// TIA Portal V17 export
// export: Created 2022-04-06T07:28:41.6787381Z, ExportSetting WithDefaults, DisplayName Totally Integrated Automation Portal, DisplayVersion V17, DisplayName TIA Portal Openness, DisplayVersion V17, DisplayName TIA Portal Version Control Interface, DisplayVersion V17, DisplayName TIA Portal Test Suite Advanced, DisplayVersion V17, DisplayName SINAMICS Startdrive Advanced, DisplayVersion V17, DisplayName SINAMICS Startdrive G130, G150, S120, S150, SINAMICS MV, S210, DisplayVersion V17, DisplayName SINAMICS Startdrive G110M, G120, G120C, G120D, G120P, G115D, DisplayVersion V17, DisplayName STEP 7 Professional, DisplayVersion V17, DisplayName STEP 7 Safety, DisplayVersion V17, DisplayName WinCC Advanced / Unified PC, DisplayVersion V17
TYPE "LAxisCtrl_typeStop"
TITLE = LAxisCtrl_typeStop
// Support: tech.team.motioncontrol@siemens.com
// stored: IsFailsafeCompliant false
   STRUCT
      deceleration : LReal := -1.0;   // Deceleration setpoint for stop (Value > 0.0: The specified value is used; Value = 0.0: Not permitted; Value < 0.0: Use of the default value configured in the technology object)
      jerk : LReal := -1.0;   // Jerk for stop (Value > 0.0: Smooth velocity profile, the specified value is used; Value = 0.0: Trapezoid velocity profile; Value < 0.0: Use of the default value configured in the technology object)
      abortAcceleration : Bool := FALSE;   // TRUE: The acceleration is set to 0.0 at the start of the job, and the deceleration immediately builds up; FALSE: The current acceleration at the start of the job is reduced using the configured jerk. Afterwards, the deceleration builds up
   END_STRUCT;
END_TYPE
